// TIA Portal V21 export
DATA_BLOCK "pulse"   // DB8
{ S7_Optimized_Access := 'FALSE' }
   VAR
      ControlKeyOff : Bool;
      EmergencyStopPressed : Bool;
      PowerReset : Bool;
      CompresseDairPressurelow : Bool;
      PowerFailure : Bool;
      PlcRestarted : Bool;
      Mm01FeedbackTrip : Bool;
      Cp01FeedbackTrip : Bool;
      Mm01OverloadTrip : Bool;
      Cp01OverloadTrip : Bool;
      MinimumWeightRequiredToStartmm01 : Bool;
      Ticr01WireBreak : Bool;
      Ticr02WireBreak : Bool;
      Ticr03WireBreak : Bool;
      Ticr04WireBreak : Bool;
      Ticr05WireBreak : Bool;
      Ticr06WireBreak : Bool;
      Ticr07WireBreak : Bool;
      Ticr08WireBreak : Bool;
      Ticr09WireBreak : Bool;
      Ticr10WireBreak : Bool;
      Picr01WireBreak : Bool;
      Picr02WireBreak : Bool;
      Picr03WireBreak : Bool;
      Picr04WireBreak : Bool;
      Cicr01WireBreak : Bool;
      Lc01CommunicationFailed : Bool;
      VesselHighPressure : Bool;
      Mm01SpeedSensorTrip : Bool;
      PlcToHmiCommunicationFailed : Bool;
      CipCycleOver : Bool;
      CipCycleConductivityReached : Bool;
      CipCycleConductivityNotReached : Bool;
      ConductivityNotSampled : Bool;
      CipReportDataNotLogged : Bool;
      PhtFailed : Bool;
      PhtPass : Bool;
      PhtOver : Bool;
      PhtReportDataNotLogged : Bool;
      SterilizationTimeOver : Bool;
      SteamFlowLow : Bool;
      SterilizationHighTemperature : Bool;
      SterilizationCycleCompleted : Bool;
      SterilizationReportDataNotLogged : Bool;
      WfiFlowLow : Bool;
      BatchReportDataNotLogged : Bool;
   END_VAR
BEGIN
END_DATA_BLOCK
